TYPE (* IEC61131-3, Table 14#5 *)
  (* Standard: 1131-3 *)
  (* Version 0.0, 1/8/2024, Cheyan, Schneider Electric, Template *)
  PACKAGE Main;
  {SET_ATTRIBUTE(nxtDataType, UylDVgj4yyHsYuYBrz+XyIF5RgwkDTRkDMdeDD9RKsv1mej6c4iFFEoDNpJc2k+xb8G7rpytc65C4Su2Rxwz5kb43Yb/BKy0)}
  SPC : STRUCT
    ctlModel : CtlModels;
  END_STRUCT;
END_TYPE
